// TIA Portal V18 export
TYPE "MEStoPLC_ResultsStoredScanExchange_ext"
// stored: IsFailsafeCompliant false
   STRUCT
      Load_ResultsStored1OK : Bool;   // Unloading part process - Results stored OK
      Load_ResultsStored1NG : Bool;   // Unloading part process - Results stored NG
      Load_ResultsStored1ReqMesDone : Bool;   // 存储完成，PLC复位 Station*DataSaveReq
      Load_ResultsStored1Spare : Bool;   // Spare
      Load_ResultsStored1Spare1 : Bool;   // Spare
      Load_ResultsStored1Spare2 : Bool;   // Spare
      Load_ResultsStored1Spare3 : Bool;   // Spare
      Load_ResultsStored1Spare4 : Bool;   // Spare
      Load_ResultsStored2OK : Bool;   // Unloading part process - Results stored OK
      Load_ResultsStored2NG : Bool;   // Unloading part process - Results stored NG
      Load_ResultsStored2ReqMesDone : Bool;   // 存储完成，PLC复位 Station*DataSaveReq
      Load_ResultsStored2Spare : Bool;   // Spare
      Load_ResultsStored2Spare1 : Bool;   // Spare
      Load_ResultsStored2Spare2 : Bool;   // Spare
      Load_ResultsStored2Spare3 : Bool;   // Spare
      Load_ResultsStored2Spare4 : Bool;   // Spare
      Load_ResultsStored3OK : Bool;   // 订单号
      Load_ResultsStored3NG : Bool;   // Unloading part process - Results stored OK
      Load_ResultsStored3ReqMesDone : Bool;   // Unloading part process - Results stored NG
      Load_ResultsStored3Spare : Bool;   // 存储完成，PLC复位 Station*DataSaveReq
      Load_ResultsStored3Spare1 : Bool;   // Spare
      Load_ResultsStored3Spare2 : Bool;   // Spare
      Load_ResultsStored3Spare3 : Bool;   // Spare
      Load_ResultsStored3Spare4 : Bool;   // Spare
      Load_ResultsStored4OK : Bool;   // Unloading part process - Results stored OK
      Load_ResultsStored4NG : Bool;   // Unloading part process - Results stored NG
      Load_ResultsStored4ReqMesDone : Bool;   // 存储完成，PLC复位 Station*DataSaveReq
      Load_ResultsStored4Spare : Bool;   // Spare
      Load_ResultsStored4Spare1 : Bool;   // Spare
      Load_ResultsStored4Spare2 : Bool;   // Spare
      Load_ResultsStored4Spare3 : Bool;   // Spare
      Load_ResultsStored4Spare4 : Bool;   // Spare
      Load_ResultsStored5OK : Bool;   // Unloading part process - Results stored OK
      Load_ResultsStored5NG : Bool;   // Unloading part process - Results stored NG
      Load_ResultsStored5ReqMesDone : Bool;   // 存储完成，PLC复位 Station*DataSaveReq
      Load_ResultsStored5Spare : Bool;   // Spare
      Load_ResultsStored5Spare1 : Bool;   // Spare
      Load_ResultsStored5Spare2 : Bool;   // Spare
      Load_ResultsStored5Spare3 : Bool;   // Spare
      Load_ResultsStored5Spare4 : Bool;   // Spare
      Load_ResultsStored6OK : Bool;   // Unloading part process - Results stored OK
      Load_ResultsStored6NG : Bool;   // Unloading part process - Results stored NG
      Load_ResultsStored6ReqMesDone : Bool;   // 存储完成，PLC复位 Station*DataSaveReq
      Load_ResultsStored6Spare : Bool;   // Spare
      Load_ResultsStored6Spare1 : Bool;   // Spare
      Load_ResultsStored6Spare2 : Bool;   // Spare
      Load_ResultsStored6Spare3 : Bool;   // Spare
      Load_ResultsStored6Spare4 : Bool;   // Spare
      Spare : Byte;   // SpareByte
      Load_ResultsStored7OK : Bool;   // Unloading part process - Results stored OK
      Load_ResultsStored7NG : Bool;   // Unloading part process - Results stored NG
      Load_ResultsStored7ReqMesDone : Bool;   // 存储完成，PLC复位 Station*DataSaveReq
      Load_ResultsStored7Spare : Bool;   // Spare
      Load_ResultsStored7Spare1 : Bool;   // Spare
      Load_ResultsStored7Spare2 : Bool;   // Spare
      Load_ResultsStored7Spare3 : Bool;   // Spare
      Load_ResultsStored7Spare4 : Bool;   // Spare
      Load_ResultsStored8OK : Bool;   // Unloading part process - Results stored OK
      Load_ResultsStored8NG : Bool;   // Unloading part process - Results stored NG
      Load_ResultsStored8ReqMesDone : Bool;   // 存储完成，PLC复位 Station*DataSaveReq
      Load_ResultsStored8Spare : Bool;   // Spare
      Load_ResultsStored8Spare5 : Bool;   // Spare
      Load_ResultsStored8Spare6 : Bool;   // Spare
      Load_ResultsStored8Spare8 : Bool;   // Spare
      Load_ResultsStored8Spare9 : Bool;   // Spare
   END_STRUCT;
END_TYPE
